(* PLC project Blank Project, Blank Blank 1.0 *)
(* stored: creationDateTime 2016-05-18T21:14:07, modificationDateTime 2017-10-06T12:31:54 *)

PROGRAM Cell2
  VAR
    C1_IR AT %IX0.3 : BOOL := true;
    M1_IR AT %IX0.4 : BOOL := true;
    Main AT %IX0.6 : BOOL := true;
    M1_motor AT %QX0.2 : BOOL := true;
    C2_motor AT %QX0.4 : BOOL := true;
  END_VAR
  VAR
    C2_working : BOOL := false;
  END_VAR
  VAR
    C2_working_int AT %MD1 : DINT := 0;
  END_VAR
  VAR
    C2_afterM : BOOL := false;
  END_VAR
  VAR
    C2_afterM_int AT %MD2 : DINT := 0;
  END_VAR
  VAR
    Step1 : BOOL := false;
  END_VAR
  VAR
    Step1_int AT %MD3 : DINT := 0;
  END_VAR
  VAR
    Step2 : BOOL := false;
  END_VAR
  VAR
    Step2_int AT %MD4 : DINT := 0;
  END_VAR
  VAR
    Step3 : BOOL := false;
  END_VAR
  VAR
    Step3_int AT %MD5 : DINT := 0;
  END_VAR
  VAR
    Pause1 : BOOL := false;
  END_VAR
  VAR
    Pause1_int AT %MD6 : DINT := 0;
  END_VAR
  VAR
    Pause2 : BOOL := false;
  END_VAR
  VAR
    Pause2_int AT %MD7 : DINT := 0;
  END_VAR
  VAR
    Timer_conveyor : TON;
    Timer_machining : TON;
    TON0 : TON;
    TON1 : TON;
    TON2 : TON;
    TON3 : TON;
    TON4 : TON;
  END_VAR
  VAR
    jadeProg1 AT %IX0.7 : BOOL := true;
  END_VAR

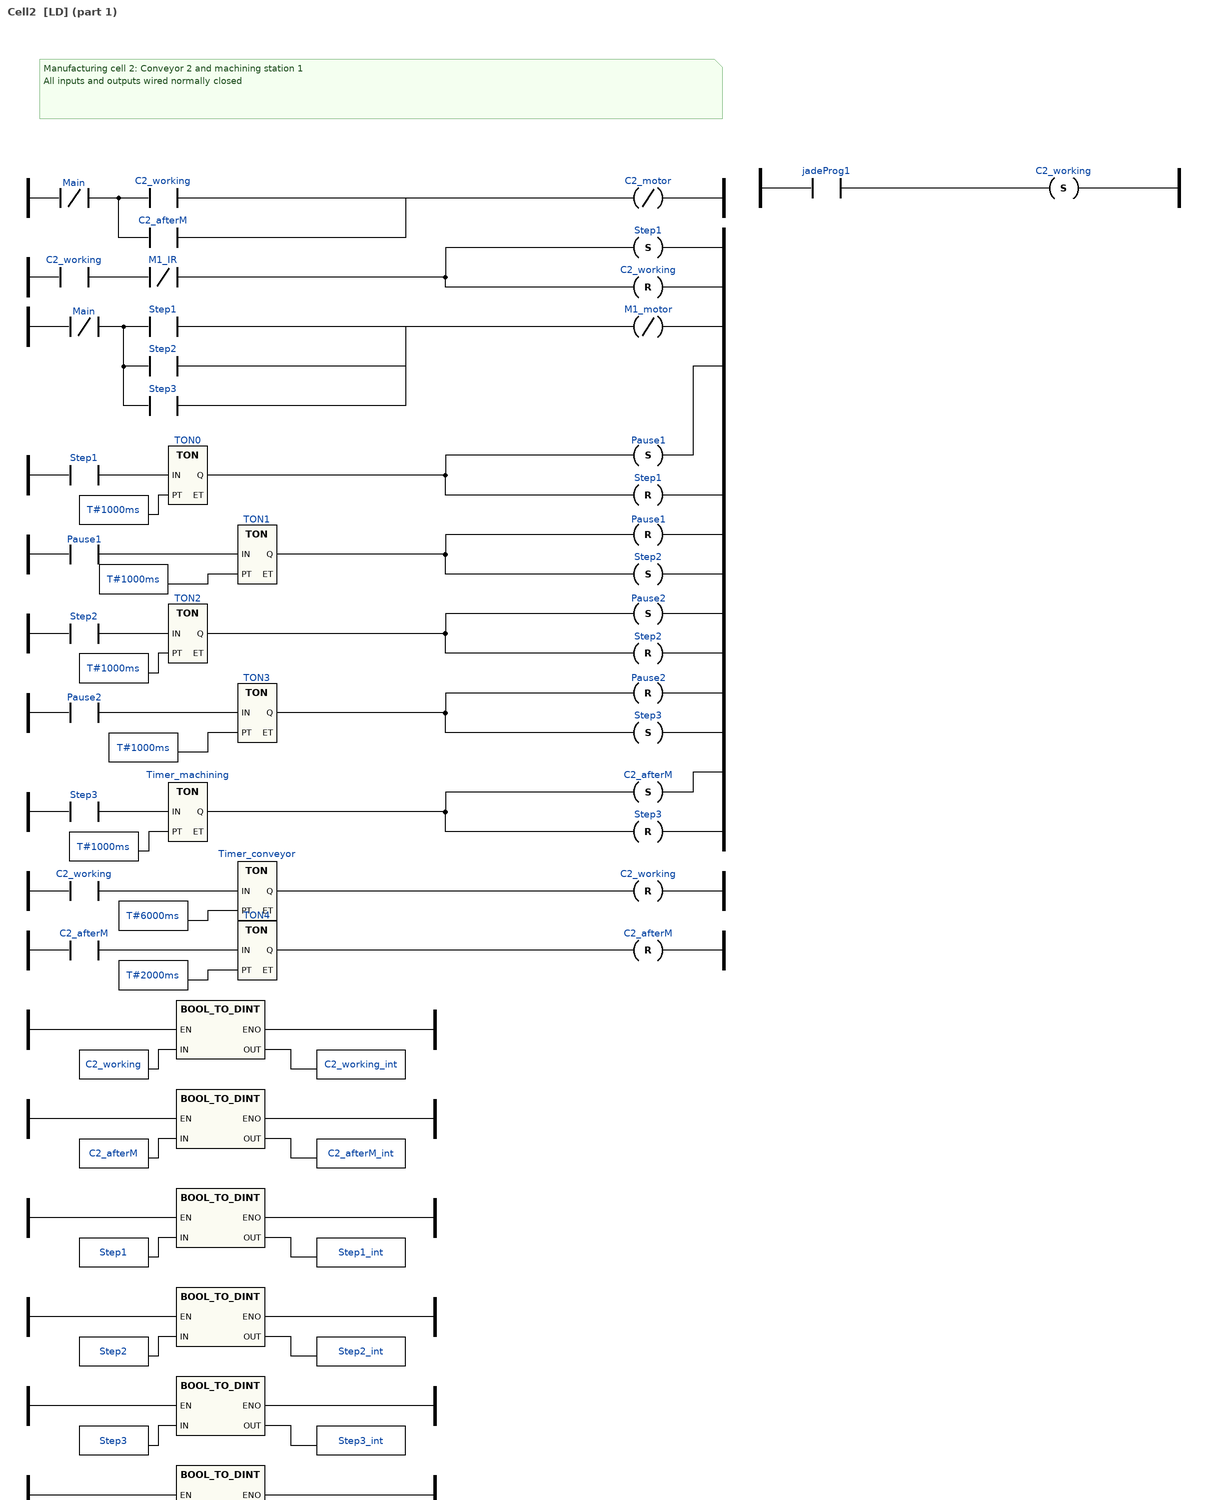
(* LD diagram, written out as Structured Text *)
(* Manufacturing cell 2: Conveyor 2 and machining station 1
All inputs and outputs wired normally closed *)
IF jadeProg1 THEN C2_working := TRUE; END_IF;
C2_motor := NOT (NOT Main AND (C2_working OR C2_afterM));
IF C2_working AND NOT M1_IR THEN Step1 := TRUE; END_IF;
IF C2_working AND NOT M1_IR THEN C2_working := FALSE; END_IF;
M1_motor := NOT (NOT Main AND (Step1 OR Step2 OR Step3));
TON0(IN := Step1, PT := T#1000ms);
IF TON0.Q THEN Pause1 := TRUE; END_IF;
IF TON0.Q THEN Step1 := FALSE; END_IF;
TON1(IN := Pause1, PT := T#1000ms);
IF TON1.Q THEN Pause1 := FALSE; END_IF;
IF TON1.Q THEN Step2 := TRUE; END_IF;
TON2(IN := Step2, PT := T#1000ms);
IF TON2.Q THEN Pause2 := TRUE; END_IF;
IF TON2.Q THEN Step2 := FALSE; END_IF;
TON3(IN := Pause2, PT := T#1000ms);
IF TON3.Q THEN Pause2 := FALSE; END_IF;
IF TON3.Q THEN Step3 := TRUE; END_IF;
Timer_machining(IN := Step3, PT := T#1000ms);
IF Timer_machining.Q THEN C2_afterM := TRUE; END_IF;
IF Timer_machining.Q THEN Step3 := FALSE; END_IF;
Timer_conveyor(IN := C2_working, PT := T#6000ms);
IF Timer_conveyor.Q THEN C2_working := FALSE; END_IF;
TON4(IN := C2_afterM, PT := T#2000ms);
IF TON4.Q THEN C2_afterM := FALSE; END_IF;
C2_working_int := BOOL_TO_DINT(C2_working);
C2_afterM_int := BOOL_TO_DINT(C2_afterM);
Step1_int := BOOL_TO_DINT(Step1);
Step2_int := BOOL_TO_DINT(Step2);
Step3_int := BOOL_TO_DINT(Step3);
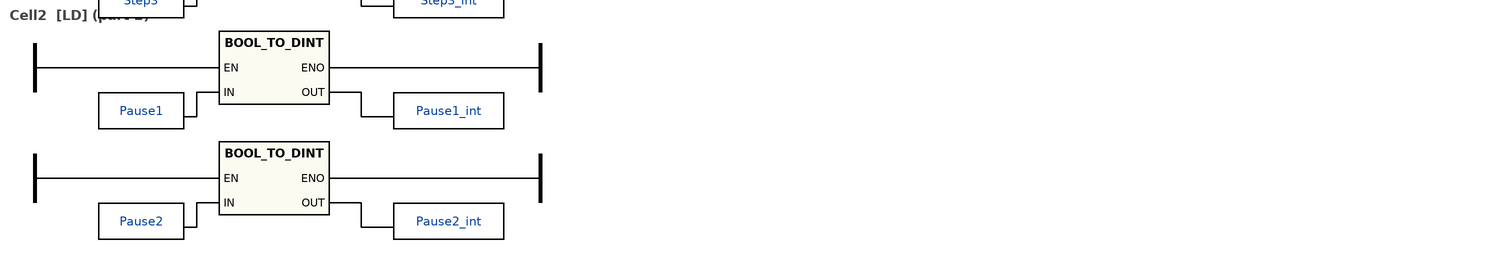
Pause1_int := BOOL_TO_DINT(Pause1);
Pause2_int := BOOL_TO_DINT(Pause2);
END_PROGRAM

CONFIGURATION Config0
  RESOURCE Res0 ON PLC
    TASK TaskMain(INTERVAL := T#50ms, PRIORITY := 0);
    PROGRAM Inst0 WITH TaskMain : Cell2;
  END_RESOURCE
END_CONFIGURATION
